TYPE ST_MOVER_SELECTOR_CTRL :
STRUCT
  Selector      : E_MOVER_SELECTOR; // select by array Index OR AXIS_REF.NcToPlc.AxisId 
  Mover         : UINT;             // array Index OR AXIS_REF.NcToPlc.AxisId
  Control       : ST_MOVER_CTRL;    // mover control struct, put motion command in here

  Data          : ST_MOVE_DATA;     // write your movement parameters
  //Gear          : ST_GEAR_DATA;     // write your gearing parameters
END_STRUCT
END_TYPE

(* stored: Version 1.1.0.1
   DUT ST_MOVER_SELECTOR_CTRL: Id {7bcabe4f-c2d6-417b-b7d0-0e7ea9cfaa6a} *)
